(* CODESYS project reflex4.project

Project tree, tasks and I/O mapping:
  Device : CODESYS Control Win V3, 3S - Smart Software Solutions GmbH, order no. 305021, version 3.5.8.10
    application Application
      libraries: Standard, * (System); BASIC, 3.31 (OSCAT)
      task MainTask (cyclic, interval t#20ms, priority 1) calls PLC_PRG
      program PLC_PRG [ST]
      visualisation Visualization
  libraries: VisuSymbols, 3.5.8.0 (System)
  text list GlobalTextList
*)

// Device/Application/PLC_PRG
PROGRAM PLC_PRG
VAR
	t1: TON;
	t2: TON;
	set: INT;
	random: BOOL := TRUE;
	start: BOOL := TRUE;
	controls: ARRAY [1..4] OF BOOL;
	switches: ARRAY [1..4] OF BOOL;
	points: ARRAY [1..15] OF BOOL;
	game: ARRAY [1..15] OF BOOL;
END_VAR

IF(start = TRUE) THEN
	random := TRUE;
	IF(random = TRUE) THEN
		start := FALSE;
		set := RDM2(last:=0,low:=1,high:=4);
	END_IF
END_IF

IF(set = 1) THEN
	random := FALSE;
	t1(IN:=TRUE,PT:=T#7000MS);
	t2(IN:=TRUE,PT:=T#2000MS);
	controls[set] := TRUE;
	IF(TIME_TO_INT(t2.ET) = 2000) THEN
 		controls[set] := FALSE;
		t2.IN := FALSE;
	END_IF
	IF((TIME_TO_INT(t1.ET) <= 7000) AND (TIME_TO_INT(t1.ET) > 2000)) THEN
		IF(switches[set] = TRUE) THEN
			points[1] := TRUE;
			switches[set] := FALSE;
			t1.IN := FALSE;
		END_IF
		IF(TIME_TO_INT(t1.ET) = 7000) THEN
			t1.IN := FALSE;
		END_IF
	END_IF
END_IF
IF(set = 2) THEN
	random := FALSE;
	t1(IN:=TRUE,PT:=T#7000MS);
	t2(IN:=TRUE,PT:=T#2000MS);
	controls[set] := TRUE;
	IF(TIME_TO_INT(t2.ET) = 2000) THEN
 		controls[set] := FALSE;
		t2.IN := FALSE;
	END_IF
	IF((TIME_TO_INT(t1.ET) <= 7000) AND (TIME_TO_INT(t1.ET) > 2000)) THEN
		IF(switches[set] = TRUE) THEN
			points[1] := TRUE;
			switches[set] := FALSE;
			t1.IN := FALSE;
		END_IF
		IF(TIME_TO_INT(t1.ET) = 7000) THEN
			t1.IN := FALSE;
		END_IF
	END_IF
END_IF
IF(set = 3) THEN
	random := FALSE;
	t1(IN:=TRUE,PT:=T#7000MS);
	t2(IN:=TRUE,PT:=T#2000MS);
	controls[set] := TRUE;
	IF(TIME_TO_INT(t2.ET) = 2000) THEN
 		controls[set] := FALSE;
		t2.IN := FALSE;
	END_IF
	IF((TIME_TO_INT(t1.ET) <= 7000) AND (TIME_TO_INT(t1.ET) > 2000)) THEN
		IF(switches[set] = TRUE) THEN
			points[1] := TRUE;
			switches[set] := FALSE;
			t1.IN := FALSE;
		END_IF
		IF(TIME_TO_INT(t1.ET) = 7000) THEN
			t1.IN := FALSE;
		END_IF
	END_IF
END_IF
IF(set = 4) THEN
	random := FALSE;
	t1(IN:=TRUE,PT:=T#7000MS);
	t2(IN:=TRUE,PT:=T#2000MS);
	controls[set] := TRUE;
	IF(TIME_TO_INT(t2.ET) = 2000) THEN
 		controls[set] := FALSE;
		t2.IN := FALSE;
	END_IF
	IF((TIME_TO_INT(t1.ET) <= 7000) AND (TIME_TO_INT(t1.ET) > 2000)) THEN
		IF(switches[set] = TRUE) THEN
			points[1] := TRUE;
			switches[set] := FALSE;
			t1.IN := FALSE;
		END_IF
		IF(TIME_TO_INT(t1.ET) = 7000) THEN
			t1.IN := FALSE;
		END_IF
	END_IF
END_IF

END_PROGRAM

// Device/Application/Visualization
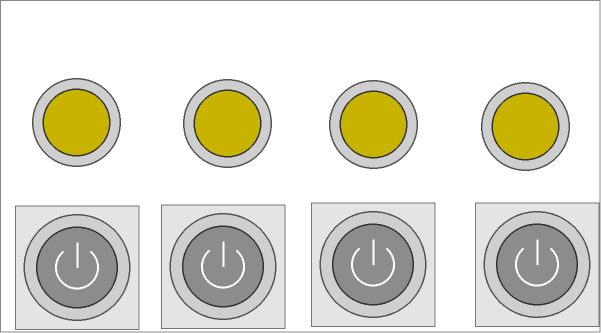
VISUALIZATION Visualization  // 601x333
    Lamp1 (25,64 103x117), variable: PLC_PRG.controls[1], style: Lamp-Lamp1-Yellow
    Lamp1 (176,65 103x117), variable: PLC_PRG.controls[2], style: Lamp-Lamp1-Yellow
    Lamp1 (322,66 103x117), variable: PLC_PRG.controls[3], style: Lamp-Lamp1-Yellow
    Lamp1 (474,68 103x117), variable: PLC_PRG.controls[4], style: Lamp-Lamp1-Yellow
    PowerSwitch (15,204 124x127), variable: PLC_PRG.switches[1], behaviour: TOGGLE, style: Switch-PowerSwitch-Gray
    PowerSwitch (161,203 124x127), variable: PLC_PRG.switches[2], behaviour: TOGGLE, style: Switch-PowerSwitch-Gray
    PowerSwitch (311,201 124x127), variable: PLC_PRG.switches[3], behaviour: TOGGLE, style: Switch-PowerSwitch-Gray
    PowerSwitch (475,201 124x127), variable: PLC_PRG.switches[4], behaviour: TOGGLE, style: Switch-PowerSwitch-Gray
END_VISUALIZATION
